FUNCTION_BLOCK FB_ToMakeSureThePLCWorks

VAR
	fbMult	: FB_Multiply2Ints;
	result	: INT;
END_VAR

fbMult(Int1 := 2, Int2 := 15, Result => result);

END_FUNCTION_BLOCK

(* stored: Version 1.1.0.1, ProductVersion 3.1.4024.12
   POU FB_ToMakeSureThePLCWorks: Id {dcf0bc4a-7d51-4eb7-8c5e-c1d67a338667}, SpecialFunc None *)
